// TwinCAT 3 PLC project Plc
// ProgramVersion: 3.1.4023.0
// libraries:
//   Tc2_Standard, * (Beckhoff Automation GmbH)
//   Tc2_System, * (Beckhoff Automation GmbH)
//   Tc3_Module, * (Beckhoff Automation GmbH)
// project tree:
//   / PlcTask.TcTTO (not stored)
//   DUTs/IO/PDOs/ InfoData_6F19DB2B.TcDUT (not stored), DeviceState_Inputs_Device_A1210598.TcDUT, DeviceState_Inputs_4751FF76.TcDUT, IO_Link_Port1_in_4EEDF10D.TcDUT, IO_Link_Port2_in_4EEDF10D.TcDUT, IO_Link_Port3_in_4EEDF10D.TcDUT, IO_Link_Port4_in_4EEDF10D.TcDUT, IO_Link_Port1_out_F2E0F4CF.TcDUT, IO_Link_Port2_out_F2E0F4CF.TcDUT, IO_Link_Port3_out_F2E0F4CF.TcDUT, IO_Link_Port4_out_F2E0F4CF.TcDUT, WcState_9091E0EB.TcDUT, InfoData_90184F0C.TcDUT, InfoData_E68C61CD.TcDUT (not stored), WcState_0B2B16F9.TcDUT (not stored), InfoData_2A97D6CF.TcDUT (not stored), Inputs_A65FACA4.TcDUT (not stored), Outputs_23C0ED1D.TcDUT (not stored)
//   DUTs/IO/Boxes/ EK1100_1FC0878B.TcDUT (not stored), EL6224_D35EF4E0.TcDUT
//   DUTs/IO/Devices/ SyncUnitTask_2D604ED5.TcDUT (not stored), SyncUnitTasks_6FEB8257.TcDUT (not stored), SyncUnits_99E584AF.TcDUT (not stored)
//   DUTs/IO/Topology/ Term_1_EK1100_9283C2D0.TcDUT (not stored), Device_1_EtherCAT_AB424CAF.TcDUT (not stored)
//   DUTs/IO/Base/ EtcSlaveBase_82538BE2.TcDUT (not stored), EtcSlaveBase_82538BE2.TcDUT (not stored), EtcSlaveBase_82538BE2.TcDUT (not stored), EtcSlaveTerminalBase_947E5A46.TcDUT (not stored), EtcSlaveBoxBase_77A0E4A7.TcDUT (not stored), EtcSlaveEndTerminalBase_866C7F0C.TcDUT (not stored), InputBase_8311D824.TcDUT (not stored), OutputBase_10CEE7DE.TcDUT (not stored), EtcMasterBase_62654B43.TcDUT (not stored)
//   GVLs/ GVL_iXlinker.TcGVL (not stored)
// real-time tasks:
//   TASK PlcTask: cycle T#10ms, priority 20, ADS port 350
// I/O:
//   DEVICE Device 1 (EtherCAT), AmsNetId 172.20.30.238.2.1
//     Term 1 (EK1100) [EK1100 EtherCAT Coupler (2A E-Bus)]
//       Term 2 (EL6224) [EL6224 (IO Link Master)]
// variable links:
//   Plc/Plc Instance <-> Device 1 (EtherCAT)/Term 1 (EK1100)
//     PlcTask Inputs/GVL_iXlinker.Device_1_EtherCAT.Term_1_EK1100.InfoData.State <-> InfoData/State
//   Plc/Plc Instance <-> Device 1 (EtherCAT)/Term 1 (EK1100)/Term 2 (EL6224)
//     PlcTask Inputs/GVL_iXlinker.Device_1_EtherCAT.Term_1_EK1100.Term_2_EL6224.DeviceState_Inputs_Device.Device_Diag <-> DeviceState Inputs Device/Device Diag
//     PlcTask Inputs/GVL_iXlinker.Device_1_EtherCAT.Term_1_EK1100.Term_2_EL6224.DeviceState_Inputs_Device.Device_State <-> DeviceState Inputs Device/Device State
//     PlcTask Inputs/GVL_iXlinker.Device_1_EtherCAT.Term_1_EK1100.Term_2_EL6224.DeviceState_Inputs.State_Ch{1..4} <-> DeviceState Inputs/State Ch{1..4}  (4 links)
//     PlcTask Inputs/GVL_iXlinker.Device_1_EtherCAT.Term_1_EK1100.Term_2_EL6224.IO_Link_Port1_in.Bitheader_1 <-> IO-Link Port1_in/Bitheader 1
//     PlcTask Inputs/GVL_iXlinker.Device_1_EtherCAT.Term_1_EK1100.Term_2_EL6224.IO_Link_Port1_in.Bitheader_2 <-> IO-Link Port1_in/Bitheader 2
//     PlcTask Inputs/GVL_iXlinker.Device_1_EtherCAT.Term_1_EK1100.Term_2_EL6224.IO_Link_Port2_in.Bitheader_1 <-> IO-Link Port2_in/Bitheader 1
//     PlcTask Inputs/GVL_iXlinker.Device_1_EtherCAT.Term_1_EK1100.Term_2_EL6224.IO_Link_Port2_in.Bitheader_2 <-> IO-Link Port2_in/Bitheader 2
//     PlcTask Inputs/GVL_iXlinker.Device_1_EtherCAT.Term_1_EK1100.Term_2_EL6224.IO_Link_Port3_in.Bitheader_1 <-> IO-Link Port3_in/Bitheader 1
//     PlcTask Inputs/GVL_iXlinker.Device_1_EtherCAT.Term_1_EK1100.Term_2_EL6224.IO_Link_Port3_in.Bitheader_2 <-> IO-Link Port3_in/Bitheader 2
//     PlcTask Inputs/GVL_iXlinker.Device_1_EtherCAT.Term_1_EK1100.Term_2_EL6224.IO_Link_Port4_in.Bitheader_1 <-> IO-Link Port4_in/Bitheader 1
//     PlcTask Inputs/GVL_iXlinker.Device_1_EtherCAT.Term_1_EK1100.Term_2_EL6224.IO_Link_Port4_in.Bitheader_2 <-> IO-Link Port4_in/Bitheader 2
//     PlcTask Inputs/GVL_iXlinker.Device_1_EtherCAT.Term_1_EK1100.Term_2_EL6224.IO_Link_Port1_in.Byte_x[0] <-> IO-Link Port1_in/Byte 1
//     PlcTask Inputs/GVL_iXlinker.Device_1_EtherCAT.Term_1_EK1100.Term_2_EL6224.IO_Link_Port1_in.Byte_x[1] <-> IO-Link Port1_in/Byte 2
//     PlcTask Inputs/GVL_iXlinker.Device_1_EtherCAT.Term_1_EK1100.Term_2_EL6224.IO_Link_Port1_in.Byte_x[2] <-> IO-Link Port1_in/Byte 3
//     PlcTask Inputs/GVL_iXlinker.Device_1_EtherCAT.Term_1_EK1100.Term_2_EL6224.IO_Link_Port1_in.Byte_x[3] <-> IO-Link Port1_in/Byte 4
//     PlcTask Inputs/GVL_iXlinker.Device_1_EtherCAT.Term_1_EK1100.Term_2_EL6224.IO_Link_Port1_in.Byte_x[4] <-> IO-Link Port1_in/Byte 5
//     PlcTask Inputs/GVL_iXlinker.Device_1_EtherCAT.Term_1_EK1100.Term_2_EL6224.IO_Link_Port1_in.Byte_x[5] <-> IO-Link Port1_in/Byte 6
//     PlcTask Inputs/GVL_iXlinker.Device_1_EtherCAT.Term_1_EK1100.Term_2_EL6224.IO_Link_Port1_in.Byte_x[6] <-> IO-Link Port1_in/Byte 7
//     PlcTask Inputs/GVL_iXlinker.Device_1_EtherCAT.Term_1_EK1100.Term_2_EL6224.IO_Link_Port1_in.Byte_x[7] <-> IO-Link Port1_in/Byte 8
//     PlcTask Inputs/GVL_iXlinker.Device_1_EtherCAT.Term_1_EK1100.Term_2_EL6224.IO_Link_Port2_in.Byte_x[0] <-> IO-Link Port2_in/Byte 1
//     PlcTask Inputs/GVL_iXlinker.Device_1_EtherCAT.Term_1_EK1100.Term_2_EL6224.IO_Link_Port2_in.Byte_x[1] <-> IO-Link Port2_in/Byte 2
//     PlcTask Inputs/GVL_iXlinker.Device_1_EtherCAT.Term_1_EK1100.Term_2_EL6224.IO_Link_Port2_in.Byte_x[2] <-> IO-Link Port2_in/Byte 3
//     PlcTask Inputs/GVL_iXlinker.Device_1_EtherCAT.Term_1_EK1100.Term_2_EL6224.IO_Link_Port2_in.Byte_x[3] <-> IO-Link Port2_in/Byte 4
//     PlcTask Inputs/GVL_iXlinker.Device_1_EtherCAT.Term_1_EK1100.Term_2_EL6224.IO_Link_Port2_in.Byte_x[4] <-> IO-Link Port2_in/Byte 5
//     PlcTask Inputs/GVL_iXlinker.Device_1_EtherCAT.Term_1_EK1100.Term_2_EL6224.IO_Link_Port2_in.Byte_x[5] <-> IO-Link Port2_in/Byte 6
//     PlcTask Inputs/GVL_iXlinker.Device_1_EtherCAT.Term_1_EK1100.Term_2_EL6224.IO_Link_Port2_in.Byte_x[6] <-> IO-Link Port2_in/Byte 7
//     PlcTask Inputs/GVL_iXlinker.Device_1_EtherCAT.Term_1_EK1100.Term_2_EL6224.IO_Link_Port2_in.Byte_x[7] <-> IO-Link Port2_in/Byte 8
//     PlcTask Inputs/GVL_iXlinker.Device_1_EtherCAT.Term_1_EK1100.Term_2_EL6224.IO_Link_Port3_in.Byte_x[0] <-> IO-Link Port3_in/Byte 1
//     PlcTask Inputs/GVL_iXlinker.Device_1_EtherCAT.Term_1_EK1100.Term_2_EL6224.IO_Link_Port3_in.Byte_x[1] <-> IO-Link Port3_in/Byte 2
//     PlcTask Inputs/GVL_iXlinker.Device_1_EtherCAT.Term_1_EK1100.Term_2_EL6224.IO_Link_Port3_in.Byte_x[2] <-> IO-Link Port3_in/Byte 3
//     PlcTask Inputs/GVL_iXlinker.Device_1_EtherCAT.Term_1_EK1100.Term_2_EL6224.IO_Link_Port3_in.Byte_x[3] <-> IO-Link Port3_in/Byte 4
//     PlcTask Inputs/GVL_iXlinker.Device_1_EtherCAT.Term_1_EK1100.Term_2_EL6224.IO_Link_Port3_in.Byte_x[4] <-> IO-Link Port3_in/Byte 5
//     PlcTask Inputs/GVL_iXlinker.Device_1_EtherCAT.Term_1_EK1100.Term_2_EL6224.IO_Link_Port3_in.Byte_x[5] <-> IO-Link Port3_in/Byte 6
//     PlcTask Inputs/GVL_iXlinker.Device_1_EtherCAT.Term_1_EK1100.Term_2_EL6224.IO_Link_Port3_in.Byte_x[6] <-> IO-Link Port3_in/Byte 7
//     PlcTask Inputs/GVL_iXlinker.Device_1_EtherCAT.Term_1_EK1100.Term_2_EL6224.IO_Link_Port3_in.Byte_x[7] <-> IO-Link Port3_in/Byte 8
//     PlcTask Inputs/GVL_iXlinker.Device_1_EtherCAT.Term_1_EK1100.Term_2_EL6224.IO_Link_Port4_in.Byte_x[0] <-> IO-Link Port4_in/Byte 1
//     PlcTask Inputs/GVL_iXlinker.Device_1_EtherCAT.Term_1_EK1100.Term_2_EL6224.IO_Link_Port4_in.Byte_x[1] <-> IO-Link Port4_in/Byte 2
//     PlcTask Inputs/GVL_iXlinker.Device_1_EtherCAT.Term_1_EK1100.Term_2_EL6224.IO_Link_Port4_in.Byte_x[2] <-> IO-Link Port4_in/Byte 3
//     PlcTask Inputs/GVL_iXlinker.Device_1_EtherCAT.Term_1_EK1100.Term_2_EL6224.IO_Link_Port4_in.Byte_x[3] <-> IO-Link Port4_in/Byte 4
//     PlcTask Inputs/GVL_iXlinker.Device_1_EtherCAT.Term_1_EK1100.Term_2_EL6224.IO_Link_Port4_in.Byte_x[4] <-> IO-Link Port4_in/Byte 5
//     PlcTask Inputs/GVL_iXlinker.Device_1_EtherCAT.Term_1_EK1100.Term_2_EL6224.IO_Link_Port4_in.Byte_x[5] <-> IO-Link Port4_in/Byte 6
//     PlcTask Inputs/GVL_iXlinker.Device_1_EtherCAT.Term_1_EK1100.Term_2_EL6224.IO_Link_Port4_in.Byte_x[6] <-> IO-Link Port4_in/Byte 7
//     PlcTask Inputs/GVL_iXlinker.Device_1_EtherCAT.Term_1_EK1100.Term_2_EL6224.IO_Link_Port4_in.Byte_x[7] <-> IO-Link Port4_in/Byte 8
//     PlcTask Outputs/GVL_iXlinker.Device_1_EtherCAT.Term_1_EK1100.Term_2_EL6224.IO_Link_Port1_out.Bitheader_1 <-> IO-Link Port1_out/Bitheader 1
//     PlcTask Outputs/GVL_iXlinker.Device_1_EtherCAT.Term_1_EK1100.Term_2_EL6224.IO_Link_Port1_out.Bitheader_2 <-> IO-Link Port1_out/Bitheader 2
//     PlcTask Outputs/GVL_iXlinker.Device_1_EtherCAT.Term_1_EK1100.Term_2_EL6224.IO_Link_Port2_out.Bitheader_1 <-> IO-Link Port2_out/Bitheader 1
//     PlcTask Outputs/GVL_iXlinker.Device_1_EtherCAT.Term_1_EK1100.Term_2_EL6224.IO_Link_Port2_out.Bitheader_2 <-> IO-Link Port2_out/Bitheader 2
//     PlcTask Outputs/GVL_iXlinker.Device_1_EtherCAT.Term_1_EK1100.Term_2_EL6224.IO_Link_Port3_out.Bitheader_1 <-> IO-Link Port3_out/Bitheader 1
//     PlcTask Outputs/GVL_iXlinker.Device_1_EtherCAT.Term_1_EK1100.Term_2_EL6224.IO_Link_Port3_out.Bitheader_2 <-> IO-Link Port3_out/Bitheader 2
//     PlcTask Outputs/GVL_iXlinker.Device_1_EtherCAT.Term_1_EK1100.Term_2_EL6224.IO_Link_Port4_out.Bitheader_1 <-> IO-Link Port4_out/Bitheader 1
//     PlcTask Outputs/GVL_iXlinker.Device_1_EtherCAT.Term_1_EK1100.Term_2_EL6224.IO_Link_Port4_out.Bitheader_2 <-> IO-Link Port4_out/Bitheader 2
//     PlcTask Outputs/GVL_iXlinker.Device_1_EtherCAT.Term_1_EK1100.Term_2_EL6224.IO_Link_Port1_out.Byte_x[0] <-> IO-Link Port1_out/Byte 1
//     PlcTask Outputs/GVL_iXlinker.Device_1_EtherCAT.Term_1_EK1100.Term_2_EL6224.IO_Link_Port1_out.Byte_x[1] <-> IO-Link Port1_out/Byte 2
//     PlcTask Outputs/GVL_iXlinker.Device_1_EtherCAT.Term_1_EK1100.Term_2_EL6224.IO_Link_Port1_out.Byte_x[2] <-> IO-Link Port1_out/Byte 3
//     PlcTask Outputs/GVL_iXlinker.Device_1_EtherCAT.Term_1_EK1100.Term_2_EL6224.IO_Link_Port1_out.Byte_x[3] <-> IO-Link Port1_out/Byte 4
//     PlcTask Outputs/GVL_iXlinker.Device_1_EtherCAT.Term_1_EK1100.Term_2_EL6224.IO_Link_Port1_out.Byte_x[4] <-> IO-Link Port1_out/Byte 5
//     PlcTask Outputs/GVL_iXlinker.Device_1_EtherCAT.Term_1_EK1100.Term_2_EL6224.IO_Link_Port1_out.Byte_x[5] <-> IO-Link Port1_out/Byte 6
//     PlcTask Outputs/GVL_iXlinker.Device_1_EtherCAT.Term_1_EK1100.Term_2_EL6224.IO_Link_Port1_out.Byte_x[6] <-> IO-Link Port1_out/Byte 7
//     PlcTask Outputs/GVL_iXlinker.Device_1_EtherCAT.Term_1_EK1100.Term_2_EL6224.IO_Link_Port1_out.Byte_x[7] <-> IO-Link Port1_out/Byte 8
//     PlcTask Outputs/GVL_iXlinker.Device_1_EtherCAT.Term_1_EK1100.Term_2_EL6224.IO_Link_Port2_out.Byte_x[0] <-> IO-Link Port2_out/Byte 1
//     PlcTask Outputs/GVL_iXlinker.Device_1_EtherCAT.Term_1_EK1100.Term_2_EL6224.IO_Link_Port2_out.Byte_x[1] <-> IO-Link Port2_out/Byte 2
//     PlcTask Outputs/GVL_iXlinker.Device_1_EtherCAT.Term_1_EK1100.Term_2_EL6224.IO_Link_Port2_out.Byte_x[2] <-> IO-Link Port2_out/Byte 3
//     PlcTask Outputs/GVL_iXlinker.Device_1_EtherCAT.Term_1_EK1100.Term_2_EL6224.IO_Link_Port2_out.Byte_x[3] <-> IO-Link Port2_out/Byte 4
//     PlcTask Outputs/GVL_iXlinker.Device_1_EtherCAT.Term_1_EK1100.Term_2_EL6224.IO_Link_Port2_out.Byte_x[4] <-> IO-Link Port2_out/Byte 5
//     PlcTask Outputs/GVL_iXlinker.Device_1_EtherCAT.Term_1_EK1100.Term_2_EL6224.IO_Link_Port2_out.Byte_x[5] <-> IO-Link Port2_out/Byte 6
//     PlcTask Outputs/GVL_iXlinker.Device_1_EtherCAT.Term_1_EK1100.Term_2_EL6224.IO_Link_Port2_out.Byte_x[6] <-> IO-Link Port2_out/Byte 7
//     PlcTask Outputs/GVL_iXlinker.Device_1_EtherCAT.Term_1_EK1100.Term_2_EL6224.IO_Link_Port2_out.Byte_x[7] <-> IO-Link Port2_out/Byte 8
//     PlcTask Outputs/GVL_iXlinker.Device_1_EtherCAT.Term_1_EK1100.Term_2_EL6224.IO_Link_Port3_out.Byte_x[0] <-> IO-Link Port3_out/Byte 1
//     PlcTask Outputs/GVL_iXlinker.Device_1_EtherCAT.Term_1_EK1100.Term_2_EL6224.IO_Link_Port3_out.Byte_x[1] <-> IO-Link Port3_out/Byte 2
//     PlcTask Outputs/GVL_iXlinker.Device_1_EtherCAT.Term_1_EK1100.Term_2_EL6224.IO_Link_Port3_out.Byte_x[2] <-> IO-Link Port3_out/Byte 3
//     PlcTask Outputs/GVL_iXlinker.Device_1_EtherCAT.Term_1_EK1100.Term_2_EL6224.IO_Link_Port3_out.Byte_x[3] <-> IO-Link Port3_out/Byte 4
//     PlcTask Outputs/GVL_iXlinker.Device_1_EtherCAT.Term_1_EK1100.Term_2_EL6224.IO_Link_Port3_out.Byte_x[4] <-> IO-Link Port3_out/Byte 5
//     PlcTask Outputs/GVL_iXlinker.Device_1_EtherCAT.Term_1_EK1100.Term_2_EL6224.IO_Link_Port3_out.Byte_x[5] <-> IO-Link Port3_out/Byte 6
//     PlcTask Outputs/GVL_iXlinker.Device_1_EtherCAT.Term_1_EK1100.Term_2_EL6224.IO_Link_Port3_out.Byte_x[6] <-> IO-Link Port3_out/Byte 7
//     PlcTask Outputs/GVL_iXlinker.Device_1_EtherCAT.Term_1_EK1100.Term_2_EL6224.IO_Link_Port3_out.Byte_x[7] <-> IO-Link Port3_out/Byte 8
//     PlcTask Outputs/GVL_iXlinker.Device_1_EtherCAT.Term_1_EK1100.Term_2_EL6224.IO_Link_Port4_out.Byte_x[0] <-> IO-Link Port4_out/Byte 1
//     PlcTask Outputs/GVL_iXlinker.Device_1_EtherCAT.Term_1_EK1100.Term_2_EL6224.IO_Link_Port4_out.Byte_x[1] <-> IO-Link Port4_out/Byte 2
//     PlcTask Outputs/GVL_iXlinker.Device_1_EtherCAT.Term_1_EK1100.Term_2_EL6224.IO_Link_Port4_out.Byte_x[2] <-> IO-Link Port4_out/Byte 3
//     PlcTask Outputs/GVL_iXlinker.Device_1_EtherCAT.Term_1_EK1100.Term_2_EL6224.IO_Link_Port4_out.Byte_x[3] <-> IO-Link Port4_out/Byte 4
//     PlcTask Outputs/GVL_iXlinker.Device_1_EtherCAT.Term_1_EK1100.Term_2_EL6224.IO_Link_Port4_out.Byte_x[4] <-> IO-Link Port4_out/Byte 5
//     PlcTask Outputs/GVL_iXlinker.Device_1_EtherCAT.Term_1_EK1100.Term_2_EL6224.IO_Link_Port4_out.Byte_x[5] <-> IO-Link Port4_out/Byte 6
//     PlcTask Outputs/GVL_iXlinker.Device_1_EtherCAT.Term_1_EK1100.Term_2_EL6224.IO_Link_Port4_out.Byte_x[6] <-> IO-Link Port4_out/Byte 7
//     PlcTask Outputs/GVL_iXlinker.Device_1_EtherCAT.Term_1_EK1100.Term_2_EL6224.IO_Link_Port4_out.Byte_x[7] <-> IO-Link Port4_out/Byte 8
//     PlcTask Inputs/GVL_iXlinker.Device_1_EtherCAT.Term_1_EK1100.Term_2_EL6224.WcState.WcState <-> WcState/WcState
//     PlcTask Inputs/GVL_iXlinker.Device_1_EtherCAT.Term_1_EK1100.Term_2_EL6224.WcState.InputToggle <-> WcState/InputToggle
//     PlcTask Inputs/GVL_iXlinker.Device_1_EtherCAT.Term_1_EK1100.Term_2_EL6224.InfoData.AdsAddr <-> InfoData/AdsAddr
//     PlcTask Inputs/GVL_iXlinker.Device_1_EtherCAT.Term_1_EK1100.Term_2_EL6224.InfoData.AoeNetId <-> InfoData/AoeNetId
//     PlcTask Inputs/GVL_iXlinker.Device_1_EtherCAT.Term_1_EK1100.Term_2_EL6224.InfoData.State <-> InfoData/State
//   Plc/Plc Instance <-> Device 1 (EtherCAT)
//     PlcTask Inputs/GVL_iXlinker.Device_1_EtherCAT.SyncUnits._default._unreferenced.WcState.WcState <-> SyncUnits/<default>/<unreferenced>/WcState/WcState
//     PlcTask Inputs/GVL_iXlinker.Device_1_EtherCAT.SyncUnits._default._unreferenced.InfoData.ObjectId <-> SyncUnits/<default>/<unreferenced>/InfoData/ObjectId
//     PlcTask Inputs/GVL_iXlinker.Device_1_EtherCAT.SyncUnits._default._unreferenced.InfoData.State <-> SyncUnits/<default>/<unreferenced>/InfoData/State
//     PlcTask Inputs/GVL_iXlinker.Device_1_EtherCAT.SyncUnits._default._unreferenced.InfoData.SlaveCount <-> SyncUnits/<default>/<unreferenced>/InfoData/SlaveCount
//     PlcTask Inputs/GVL_iXlinker.Device_1_EtherCAT.SyncUnits._default.PlcTask.WcState.WcState <-> SyncUnits/<default>/PlcTask/WcState/WcState
//     PlcTask Inputs/GVL_iXlinker.Device_1_EtherCAT.SyncUnits._default.PlcTask.InfoData.ObjectId <-> SyncUnits/<default>/PlcTask/InfoData/ObjectId
//     PlcTask Inputs/GVL_iXlinker.Device_1_EtherCAT.SyncUnits._default.PlcTask.InfoData.State <-> SyncUnits/<default>/PlcTask/InfoData/State
//     PlcTask Inputs/GVL_iXlinker.Device_1_EtherCAT.SyncUnits._default.PlcTask.InfoData.SlaveCount <-> SyncUnits/<default>/PlcTask/InfoData/SlaveCount
//     PlcTask Inputs/GVL_iXlinker.Device_1_EtherCAT.Inputs.SlaveCount <-> Inputs/SlaveCount
//     PlcTask Inputs/GVL_iXlinker.Device_1_EtherCAT.Inputs.DevState <-> Inputs/DevState
//     PlcTask Inputs/GVL_iXlinker.Device_1_EtherCAT.Inputs.Frm0State <-> Inputs/Frm0State
//     PlcTask Inputs/GVL_iXlinker.Device_1_EtherCAT.Inputs.Frm0WcState <-> Inputs/Frm0WcState
//     PlcTask Inputs/GVL_iXlinker.Device_1_EtherCAT.Inputs.Frm0InputToggle <-> Inputs/Frm0InputToggle
//     PlcTask Outputs/GVL_iXlinker.Device_1_EtherCAT.Outputs.DevCtrl <-> Outputs/DevCtrl
//     PlcTask Outputs/GVL_iXlinker.Device_1_EtherCAT.Outputs.Frm0Ctrl <-> Outputs/Frm0Ctrl
//     PlcTask Outputs/GVL_iXlinker.Device_1_EtherCAT.Outputs.Frm0WcCtrl <-> Outputs/Frm0WcCtrl
//     PlcTask Inputs/GVL_iXlinker.Device_1_EtherCAT.InfoData.ChangeCount <-> InfoData/ChangeCount
//     PlcTask Inputs/GVL_iXlinker.Device_1_EtherCAT.InfoData.DevId <-> InfoData/DevId
//     PlcTask Inputs/GVL_iXlinker.Device_1_EtherCAT.InfoData.AmsNetId <-> InfoData/AmsNetId
//     PlcTask Inputs/GVL_iXlinker.Device_1_EtherCAT.InfoData.CfgSlaveCount <-> InfoData/CfgSlaveCount
//     PlcTask Inputs/GVL_iXlinker.Device_1_EtherCAT.InfoData.DcToTcTimeOffset <-> InfoData/DcToTcTimeOffset
//     PlcTask Inputs/GVL_iXlinker.Device_1_EtherCAT.InfoData.DcToExtTimeOffset <-> InfoData/DcToExtTimeOffset

// ---- DUTs/IO/PDOs/DeviceState_Inputs_Device_A1210598.TcDUT
{attribute 'GeneratedUsingTerminal: EL6224-0000-0021'}
{attribute addProperty BoxType "EL6224-0000-0021"}
{attribute addProperty Id "Device_DiagAT %I*BOOL1Device_StateAT %I*BOOL1"}
{attribute addProperty CRC "2703295896"}
{attribute addProperty Size "2"}
TYPE DeviceState_Inputs_Device_A1210598 EXTENDS InputBase_8311D824 :
STRUCT
	{attribute addProperty Name "Device_Diag"}
	Device_Diag AT %I* : BOOL;
	{attribute addProperty Name "Device_State"}
	Device_State AT %I* : BOOL;
END_STRUCT
END_TYPE

// ---- DUTs/IO/PDOs/DeviceState_Inputs_4751FF76.TcDUT
{attribute 'GeneratedUsingTerminal: EL6224-0000-0021'}
{attribute addProperty BoxType "EL6224-0000-0021"}
{attribute addProperty Id "State_Ch1AT %I*USINT1State_Ch2AT %I*USINT1State_Ch3AT %I*USINT1State_Ch4AT %I*USINT1"}
{attribute addProperty CRC "1196556150"}
{attribute addProperty Size "4"}
TYPE DeviceState_Inputs_4751FF76 EXTENDS InputBase_8311D824 :
STRUCT
	{attribute addProperty Name "State_Ch1"}
	State_Ch1 AT %I* : USINT;
	{attribute addProperty Name "State_Ch2"}
	State_Ch2 AT %I* : USINT;
	{attribute addProperty Name "State_Ch3"}
	State_Ch3 AT %I* : USINT;
	{attribute addProperty Name "State_Ch4"}
	State_Ch4 AT %I* : USINT;
END_STRUCT
END_TYPE

// ---- DUTs/IO/PDOs/IO_Link_Port1_in_4EEDF10D.TcDUT
{attribute 'GeneratedUsingTerminal: EL6224-0000-0021'}
{attribute addProperty BoxType "EL6224-0000-0021"}
{attribute addProperty Id "Bitheader_1AT %I*BYTE1Byte_xAT %I*ARRAY[0..7] OF BYTE8Bitheader_2AT %I*BYTE1"}
{attribute addProperty CRC "50343685"}
{attribute addProperty Size "10"}
TYPE IO_Link_Port1_in_4EEDF10D EXTENDS InputBase_8311D824 :
STRUCT
	{attribute addProperty Name "Bitheader_1"}
	Bitheader_1 AT %I* : BYTE;
	{attribute addProperty Name "Byte"}
	Byte_x AT %I* : ARRAY[0..7] OF BYTE;
	{attribute addProperty Name "Bitheader_2"}
	Bitheader_2 AT %I* : BYTE;
END_STRUCT
END_TYPE

// ---- DUTs/IO/PDOs/IO_Link_Port2_in_4EEDF10D.TcDUT
{attribute 'GeneratedUsingTerminal: EL6224-0000-0021'}
{attribute addProperty BoxType "EL6224-0000-0021"}
{attribute addProperty Id "Bitheader_1AT %I*BYTE1Byte_xAT %I*ARRAY[0..7] OF BYTE8Bitheader_2AT %I*BYTE1"}
{attribute addProperty CRC "50343685"}
{attribute addProperty Size "10"}
TYPE IO_Link_Port2_in_4EEDF10D EXTENDS InputBase_8311D824 :
STRUCT
	{attribute addProperty Name "Bitheader_1"}
	Bitheader_1 AT %I* : BYTE;
	{attribute addProperty Name "Byte"}
	Byte_x AT %I* : ARRAY[0..7] OF BYTE;
	{attribute addProperty Name "Bitheader_2"}
	Bitheader_2 AT %I* : BYTE;
END_STRUCT
END_TYPE

// ---- DUTs/IO/PDOs/IO_Link_Port3_in_4EEDF10D.TcDUT
{attribute 'GeneratedUsingTerminal: EL6224-0000-0021'}
{attribute addProperty BoxType "EL6224-0000-0021"}
{attribute addProperty Id "Bitheader_1AT %I*BYTE1Byte_xAT %I*ARRAY[0..7] OF BYTE8Bitheader_2AT %I*BYTE1"}
{attribute addProperty CRC "50343685"}
{attribute addProperty Size "10"}
TYPE IO_Link_Port3_in_4EEDF10D EXTENDS InputBase_8311D824 :
STRUCT
	{attribute addProperty Name "Bitheader_1"}
	Bitheader_1 AT %I* : BYTE;
	{attribute addProperty Name "Byte"}
	Byte_x AT %I* : ARRAY[0..7] OF BYTE;
	{attribute addProperty Name "Bitheader_2"}
	Bitheader_2 AT %I* : BYTE;
END_STRUCT
END_TYPE

// ---- DUTs/IO/PDOs/IO_Link_Port4_in_4EEDF10D.TcDUT
{attribute 'GeneratedUsingTerminal: EL6224-0000-0021'}
{attribute addProperty BoxType "EL6224-0000-0021"}
{attribute addProperty Id "Bitheader_1AT %I*BYTE1Byte_xAT %I*ARRAY[0..7] OF BYTE8Bitheader_2AT %I*BYTE1"}
{attribute addProperty CRC "50343685"}
{attribute addProperty Size "10"}
TYPE IO_Link_Port4_in_4EEDF10D EXTENDS InputBase_8311D824 :
STRUCT
	{attribute addProperty Name "Bitheader_1"}
	Bitheader_1 AT %I* : BYTE;
	{attribute addProperty Name "Byte"}
	Byte_x AT %I* : ARRAY[0..7] OF BYTE;
	{attribute addProperty Name "Bitheader_2"}
	Bitheader_2 AT %I* : BYTE;
END_STRUCT
END_TYPE

// ---- DUTs/IO/PDOs/IO_Link_Port1_out_F2E0F4CF.TcDUT
{attribute 'GeneratedUsingTerminal: EL6224-0000-0021'}
{attribute addProperty BoxType "EL6224-0000-0021"}
{attribute addProperty Id "Bitheader_1AT %Q*BYTE1Byte_xAT %Q*ARRAY[0..7] OF BYTE8Bitheader_2AT %Q*BYTE1"}
{attribute addProperty CRC "2855058970"}
{attribute addProperty Size "10"}
TYPE IO_Link_Port1_out_F2E0F4CF EXTENDS OutputBase_10CEE7DE :
STRUCT
	{attribute addProperty Name "Bitheader_1"}
	Bitheader_1 AT %Q* : BYTE;
	{attribute addProperty Name "Byte"}
	Byte_x AT %Q* : ARRAY[0..7] OF BYTE;
	{attribute addProperty Name "Bitheader_2"}
	Bitheader_2 AT %Q* : BYTE;
END_STRUCT
END_TYPE

// ---- DUTs/IO/PDOs/IO_Link_Port2_out_F2E0F4CF.TcDUT
{attribute 'GeneratedUsingTerminal: EL6224-0000-0021'}
{attribute addProperty BoxType "EL6224-0000-0021"}
{attribute addProperty Id "Bitheader_1AT %Q*BYTE1Byte_xAT %Q*ARRAY[0..7] OF BYTE8Bitheader_2AT %Q*BYTE1"}
{attribute addProperty CRC "2855058970"}
{attribute addProperty Size "10"}
TYPE IO_Link_Port2_out_F2E0F4CF EXTENDS OutputBase_10CEE7DE :
STRUCT
	{attribute addProperty Name "Bitheader_1"}
	Bitheader_1 AT %Q* : BYTE;
	{attribute addProperty Name "Byte"}
	Byte_x AT %Q* : ARRAY[0..7] OF BYTE;
	{attribute addProperty Name "Bitheader_2"}
	Bitheader_2 AT %Q* : BYTE;
END_STRUCT
END_TYPE

// ---- DUTs/IO/PDOs/IO_Link_Port3_out_F2E0F4CF.TcDUT
{attribute 'GeneratedUsingTerminal: EL6224-0000-0021'}
{attribute addProperty BoxType "EL6224-0000-0021"}
{attribute addProperty Id "Bitheader_1AT %Q*BYTE1Byte_xAT %Q*ARRAY[0..7] OF BYTE8Bitheader_2AT %Q*BYTE1"}
{attribute addProperty CRC "2855058970"}
{attribute addProperty Size "10"}
TYPE IO_Link_Port3_out_F2E0F4CF EXTENDS OutputBase_10CEE7DE :
STRUCT
	{attribute addProperty Name "Bitheader_1"}
	Bitheader_1 AT %Q* : BYTE;
	{attribute addProperty Name "Byte"}
	Byte_x AT %Q* : ARRAY[0..7] OF BYTE;
	{attribute addProperty Name "Bitheader_2"}
	Bitheader_2 AT %Q* : BYTE;
END_STRUCT
END_TYPE

// ---- DUTs/IO/PDOs/IO_Link_Port4_out_F2E0F4CF.TcDUT
{attribute 'GeneratedUsingTerminal: EL6224-0000-0021'}
{attribute addProperty BoxType "EL6224-0000-0021"}
{attribute addProperty Id "Bitheader_1AT %Q*BYTE1Byte_xAT %Q*ARRAY[0..7] OF BYTE8Bitheader_2AT %Q*BYTE1"}
{attribute addProperty CRC "2855058970"}
{attribute addProperty Size "10"}
TYPE IO_Link_Port4_out_F2E0F4CF EXTENDS OutputBase_10CEE7DE :
STRUCT
	{attribute addProperty Name "Bitheader_1"}
	Bitheader_1 AT %Q* : BYTE;
	{attribute addProperty Name "Byte"}
	Byte_x AT %Q* : ARRAY[0..7] OF BYTE;
	{attribute addProperty Name "Bitheader_2"}
	Bitheader_2 AT %Q* : BYTE;
END_STRUCT
END_TYPE

// ---- DUTs/IO/PDOs/WcState_9091E0EB.TcDUT
{attribute 'GeneratedUsingTerminal: EL6224-0000-0021'}
{attribute addProperty BoxType "EL6224-0000-0021"}
{attribute addProperty Id "WcStateAT %I*BOOL1InputToggleAT %I*BOOL1"}
{attribute addProperty CRC "2425479403"}
{attribute addProperty Size "2"}
TYPE WcState_9091E0EB :
STRUCT
	{attribute addProperty Name "WcState"}
	WcState AT %I* : BOOL;
	{attribute addProperty Name "InputToggle"}
	InputToggle AT %I* : BOOL;
END_STRUCT
END_TYPE

// ---- DUTs/IO/PDOs/InfoData_90184F0C.TcDUT
{attribute 'GeneratedUsingTerminal: EL6224-0000-0021'}
{attribute addProperty BoxType "EL6224-0000-0021"}
{attribute addProperty Id "AdsAddrAT %I*AMSADDR8AoeNetIdAT %I*AMSNETID6StateAT %I*UINT2"}
{attribute addProperty CRC "2417512204"}
{attribute addProperty Size "16"}
TYPE InfoData_90184F0C EXTENDS InputBase_8311D824 :
STRUCT
	{attribute addProperty Name "AdsAddr"}
	AdsAddr AT %I* : AMSADDR;
	{attribute addProperty Name "AoeNetId"}
	AoeNetId AT %I* : AMSNETID;
	{attribute addProperty Name "State"}
	State AT %I* : UINT;
END_STRUCT
END_TYPE

// ---- DUTs/IO/Boxes/EL6224_D35EF4E0.TcDUT
{attribute 'GeneratedUsingTerminal: EL6224-0000-0021'}
{attribute addProperty BoxType "EL6224-0000-0021"}
{attribute addProperty Description "EL6224 (IO Link Master)"}
{attribute addProperty Physics "KK"}
{attribute addProperty Id "DeviceState_Inputs_DeviceAT %I*DeviceState_Inputs_Device_A12105982DeviceState_InputsAT %I*DeviceState_Inputs_4751FF764IO_Link_Port1_inAT %I*IO_Link_Port1_in_4EEDF10D10IO_Link_Port2_inAT %I*IO_Link_Port2_in_4EEDF10D10IO_Link_Port3_inAT %I*IO_Link_Port3_in_4EEDF10D10IO_Link_Port4_inAT %I*IO_Link_Port4_in_4EEDF10D10IO_Link_Port1_outAT %Q*IO_Link_Port1_out_F2E0F4CF10IO_Link_Port2_outAT %Q*IO_Link_Port2_out_F2E0F4CF10IO_Link_Port3_outAT %Q*IO_Link_Port3_out_F2E0F4CF10IO_Link_Port4_outAT %Q*IO_Link_Port4_out_F2E0F4CF10WcStateAT %I*WcState_9091E0EB2InfoDataAT %I*InfoData_90184F0C16"}
{attribute addProperty CRC "3546215648"}
{attribute addProperty Size "104"}
TYPE EL6224_D35EF4E0 EXTENDS EtcSlaveTerminalBase_947E5A46 :
STRUCT
	{attribute addProperty Name "DeviceState_Inputs_Device"}
	DeviceState_Inputs_Device : DeviceState_Inputs_Device_A1210598;
	{attribute addProperty Name "DeviceState_Inputs"}
	DeviceState_Inputs : DeviceState_Inputs_4751FF76;
	{attribute addProperty Name "IO_Link_Port1_in"}
	IO_Link_Port1_in : IO_Link_Port1_in_4EEDF10D;
	{attribute addProperty Name "IO_Link_Port2_in"}
	IO_Link_Port2_in : IO_Link_Port2_in_4EEDF10D;
	{attribute addProperty Name "IO_Link_Port3_in"}
	IO_Link_Port3_in : IO_Link_Port3_in_4EEDF10D;
	{attribute addProperty Name "IO_Link_Port4_in"}
	IO_Link_Port4_in : IO_Link_Port4_in_4EEDF10D;
	{attribute addProperty Name "IO_Link_Port1_out"}
	IO_Link_Port1_out : IO_Link_Port1_out_F2E0F4CF;
	{attribute addProperty Name "IO_Link_Port2_out"}
	IO_Link_Port2_out : IO_Link_Port2_out_F2E0F4CF;
	{attribute addProperty Name "IO_Link_Port3_out"}
	IO_Link_Port3_out : IO_Link_Port3_out_F2E0F4CF;
	{attribute addProperty Name "IO_Link_Port4_out"}
	IO_Link_Port4_out : IO_Link_Port4_out_F2E0F4CF;
	{attribute addProperty Name "WcState"}
	WcState : WcState_9091E0EB;
	{attribute addProperty Name "InfoData"}
	InfoData : InfoData_90184F0C;
END_STRUCT
END_TYPE
